% RSLogix 500 project Conveyor Belt with Order Fullfillment.RSS, saved by version 8.30.00.16 %
PROJECT "UNTITLED"    % processor: Bul.1763 MicroLogix 1100 Series B %

PROGRAM FILES
  LAD 2 "MAIN"  6 rungs
  LAD 3 "INPUTS"  7 rungs
  LAD 4 "OUTPUTS"  4 rungs
  LAD 5 "CONTROLS"  16 rungs

DATA FILES
  O0 OUTPUT  4 elements
  I1 INPUT  6 elements
  S2 STATUS  66 elements
  B3 BINARY  2 elements
  T4 TIMER  3 elements
  C5 COUNTER  1 elements
  R6 CONTROL  1 elements
  N7 INTEGER  3 elements
  F8 FLOAT  1 elements

LADDER 2 "MAIN"
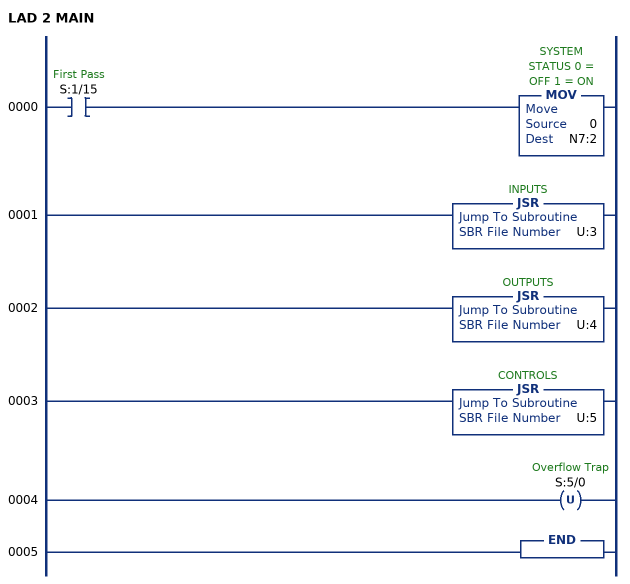
% Rung: 0 %
SOR XIC S:1/15 MOV 0 N7:2 EOR
%   S:1/15  "First Pass" %
%   N7:2  "SYSTEM STATUS 0 = OFF 1 = ON" %
% Rung: 1 %
SOR JSR U:3 EOR
%   U:3  "INPUTS" %
% Rung: 2 %
SOR JSR U:4 EOR
%   U:4  "OUTPUTS" %
% Rung: 3 %
SOR JSR U:5 EOR
%   U:5  "CONTROLS" %
% Rung: 4 %
SOR OTU S:5/0 EOR
%   S:5/0  "Overflow Trap" %
% Rung: 5 %
SOR END EOR

LADDER 3 "INPUTS"
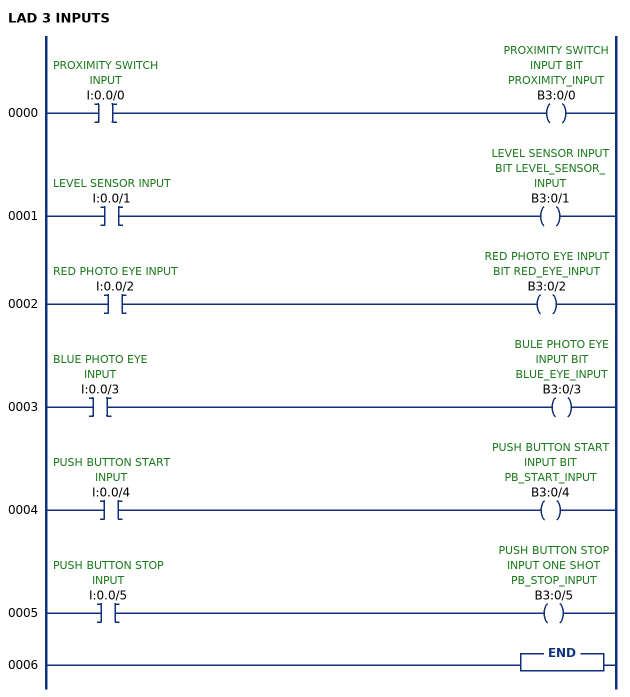
% Rung: 0 %
SOR XIC I:0.0/0 OTE B3:0/0 EOR
%   I:0.0/0  "PROXIMITY SWITCH INPUT" %
%   B3:0/0  PROXIMITY_INPUT  "PROXIMITY SWITCH INPUT BIT" %
% Rung: 1 %
SOR XIC I:0.0/1 OTE B3:0/1 EOR
%   I:0.0/1  "LEVEL SENSOR INPUT" %
%   B3:0/1  LEVEL_SENSOR_INPUT  "LEVEL SENSOR INPUT BIT" %
% Rung: 2 %
SOR XIC I:0.0/2 OTE B3:0/2 EOR
%   I:0.0/2  "RED PHOTO EYE INPUT" %
%   B3:0/2  RED_EYE_INPUT  "RED PHOTO EYE INPUT BIT" %
% Rung: 3 %
SOR XIC I:0.0/3 OTE B3:0/3 EOR
%   I:0.0/3  "BLUE PHOTO EYE INPUT" %
%   B3:0/3  BLUE_EYE_INPUT  "BULE PHOTO EYE INPUT BIT" %
% Rung: 4 %
SOR XIC I:0.0/4 OTE B3:0/4 EOR
%   I:0.0/4  "PUSH BUTTON START INPUT" %
%   B3:0/4  PB_START_INPUT  "PUSH BUTTON START INPUT BIT" %
% Rung: 5 %
SOR XIC I:0.0/5 OTE B3:0/5 EOR
%   I:0.0/5  "PUSH BUTTON STOP INPUT" %
%   B3:0/5  PB_STOP_INPUT  "PUSH BUTTON STOP INPUT ONE SHOT" %
% Rung: 6 %
SOR END EOR

LADDER 4 "OUTPUTS"
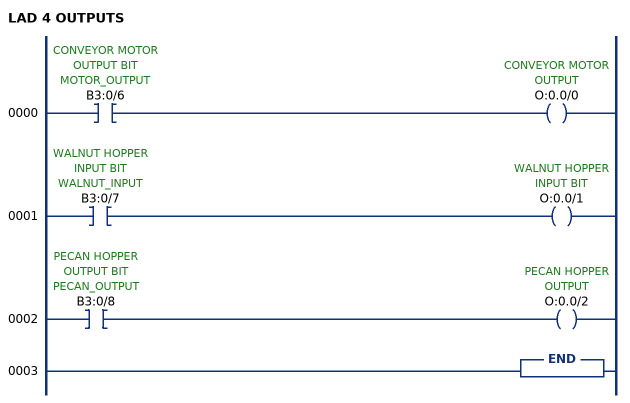
% Rung: 0 %
SOR XIC B3:0/6 OTE O:0.0/0 EOR
%   B3:0/6  MOTOR_OUTPUT  "CONVEYOR MOTOR OUTPUT BIT" %
%   O:0.0/0  "CONVEYOR MOTOR OUTPUT" %
% Rung: 1 %
SOR XIC B3:0/7 OTE O:0.0/1 EOR
%   B3:0/7  WALNUT_INPUT  "WALNUT HOPPER INPUT BIT" %
%   O:0.0/1  "WALNUT HOPPER INPUT BIT" %
% Rung: 2 %
SOR XIC B3:0/8 OTE O:0.0/2 EOR
%   B3:0/8  PECAN_OUTPUT  "PECAN HOPPER OUTPUT BIT" %
%   O:0.0/2  "PECAN HOPPER OUTPUT" %
% Rung: 3 %
SOR END EOR

LADDER 5 "CONTROLS"
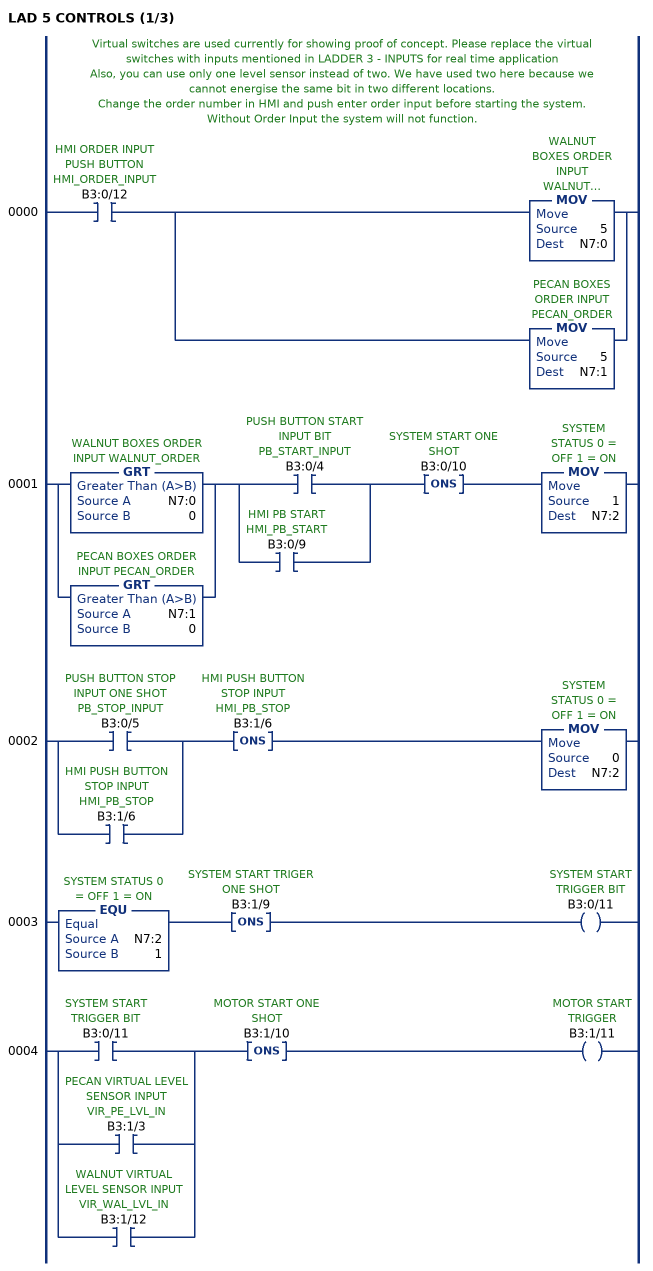
% Rung: 0 %
% Virtual switches are used currently for showing proof of concept. Please replace the virtual switches with inputs mentioned in LADDER 3 - INPUTS for real time application
% Also, you can use only one level sensor instead of two. We have used two here because we cannot energise the same bit in two different locations.
% 
% Change the order number in HMI and push enter order input before starting the system. Without Order Input the system will not function. %
SOR XIC B3:0/12 BST MOV 5 N7:0 NXB MOV 5 N7:1 BND EOR
%   B3:0/12  HMI_ORDER_INPUT  "HMI ORDER INPUT PUSH BUTTON" %
%   N7:0  WALNUT_ORDER  "WALNUT BOXES ORDER INPUT" %
%   N7:1  PECAN_ORDER  "PECAN BOXES ORDER INPUT" %
% Rung: 1 %
SOR BST GRT N7:0 0 NXB GRT N7:1 0 BND BST XIC B3:0/4 NXB XIC B3:0/9 BND ONS B3:0/10 MOV 1 N7:2 EOR
%   N7:0  WALNUT_ORDER  "WALNUT BOXES ORDER INPUT" %
%   N7:1  PECAN_ORDER  "PECAN BOXES ORDER INPUT" %
%   B3:0/4  PB_START_INPUT  "PUSH BUTTON START INPUT BIT" %
%   B3:0/9  HMI_PB_START  "HMI PB START" %
%   B3:0/10  "SYSTEM START ONE SHOT" %
%   N7:2  "SYSTEM STATUS 0 = OFF 1 = ON" %
% Rung: 2 %
SOR BST XIC B3:0/5 NXB XIC B3:1/6 BND ONS B3:1/6 MOV 0 N7:2 EOR
%   B3:0/5  PB_STOP_INPUT  "PUSH BUTTON STOP INPUT ONE SHOT" %
%   B3:1/6  HMI_PB_STOP  "HMI PUSH BUTTON STOP INPUT" %
%   N7:2  "SYSTEM STATUS 0 = OFF 1 = ON" %
% Rung: 3 %
SOR EQU N7:2 1 ONS B3:1/9 OTE B3:0/11 EOR
%   N7:2  "SYSTEM STATUS 0 = OFF 1 = ON" %
%   B3:1/9  "SYSTEM START TRIGER ONE SHOT" %
%   B3:0/11  "SYSTEM START TRIGGER BIT" %
% Rung: 4 %
SOR BST XIC B3:0/11 NXB XIC B3:1/3 NXB XIC B3:1/12 BND ONS B3:1/10 OTE B3:1/11 EOR
%   B3:0/11  "SYSTEM START TRIGGER BIT" %
%   B3:1/3  VIR_PE_LVL_IN  "PECAN VIRTUAL LEVEL SENSOR INPUT" %
%   B3:1/12  VIR_WAL_LVL_IN  "WALNUT VIRTUAL LEVEL SENSOR INPUT" %
%   B3:1/10  "MOTOR START ONE SHOT" %
%   B3:1/11  "MOTOR START TRIGGER" %

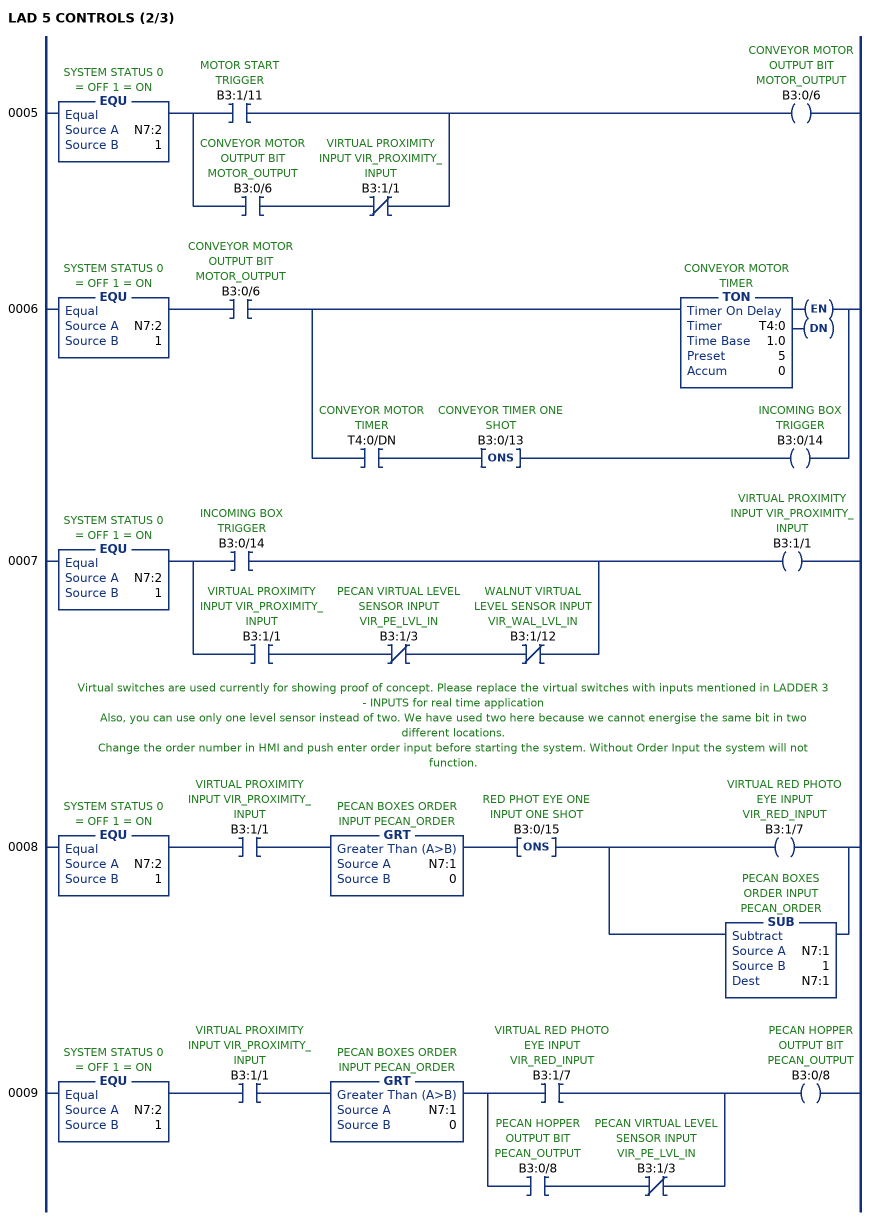
% Rung: 5 %
SOR EQU N7:2 1 BST XIC B3:1/11 NXB XIC B3:0/6 XIO B3:1/1 BND OTE B3:0/6 EOR
%   N7:2  "SYSTEM STATUS 0 = OFF 1 = ON" %
%   B3:1/11  "MOTOR START TRIGGER" %
%   B3:0/6  MOTOR_OUTPUT  "CONVEYOR MOTOR OUTPUT BIT" %
%   B3:1/1  VIR_PROXIMITY_INPUT  "VIRTUAL PROXIMITY INPUT" %
% Rung: 6 %
SOR EQU N7:2 1 XIC B3:0/6 BST TON T4:0 1.0 5 0 NXB XIC T4:0/DN ONS B3:0/13 OTE B3:0/14 BND EOR
%   N7:2  "SYSTEM STATUS 0 = OFF 1 = ON" %
%   B3:0/6  MOTOR_OUTPUT  "CONVEYOR MOTOR OUTPUT BIT" %
%   T4:0  "CONVEYOR MOTOR TIMER" %
%   B3:0/13  "CONVEYOR TIMER ONE SHOT" %
%   B3:0/14  "INCOMING BOX TRIGGER" %
% Rung: 7 %
SOR EQU N7:2 1 BST XIC B3:0/14 NXB XIC B3:1/1 XIO B3:1/3 XIO B3:1/12 BND OTE B3:1/1 EOR
%   N7:2  "SYSTEM STATUS 0 = OFF 1 = ON" %
%   B3:0/14  "INCOMING BOX TRIGGER" %
%   B3:1/1  VIR_PROXIMITY_INPUT  "VIRTUAL PROXIMITY INPUT" %
%   B3:1/3  VIR_PE_LVL_IN  "PECAN VIRTUAL LEVEL SENSOR INPUT" %
%   B3:1/12  VIR_WAL_LVL_IN  "WALNUT VIRTUAL LEVEL SENSOR INPUT" %
% Rung: 8 %
% Virtual switches are used currently for showing proof of concept. Please replace the virtual switches with inputs mentioned in LADDER 3 - INPUTS for real time application
% Also, you can use only one level sensor instead of two. We have used two here because we cannot energise the same bit in two different locations.
% 
% Change the order number in HMI and push enter order input before starting the system. Without Order Input the system will not function. %
SOR EQU N7:2 1 XIC B3:1/1 GRT N7:1 0 ONS B3:0/15 BST OTE B3:1/7 NXB SUB N7:1 1 N7:1 BND EOR
%   N7:2  "SYSTEM STATUS 0 = OFF 1 = ON" %
%   B3:1/1  VIR_PROXIMITY_INPUT  "VIRTUAL PROXIMITY INPUT" %
%   N7:1  PECAN_ORDER  "PECAN BOXES ORDER INPUT" %
%   B3:0/15  "RED PHOT EYE ONE INPUT ONE SHOT" %
%   B3:1/7  VIR_RED_INPUT  "VIRTUAL RED PHOTO EYE INPUT" %
% Rung: 9 %
SOR EQU N7:2 1 XIC B3:1/1 GRT N7:1 0 BST XIC B3:1/7 NXB XIC B3:0/8 XIO B3:1/3 BND OTE B3:0/8 EOR
%   N7:2  "SYSTEM STATUS 0 = OFF 1 = ON" %
%   B3:1/1  VIR_PROXIMITY_INPUT  "VIRTUAL PROXIMITY INPUT" %
%   N7:1  PECAN_ORDER  "PECAN BOXES ORDER INPUT" %
%   B3:1/7  VIR_RED_INPUT  "VIRTUAL RED PHOTO EYE INPUT" %
%   B3:0/8  PECAN_OUTPUT  "PECAN HOPPER OUTPUT BIT" %
%   B3:1/3  VIR_PE_LVL_IN  "PECAN VIRTUAL LEVEL SENSOR INPUT" %

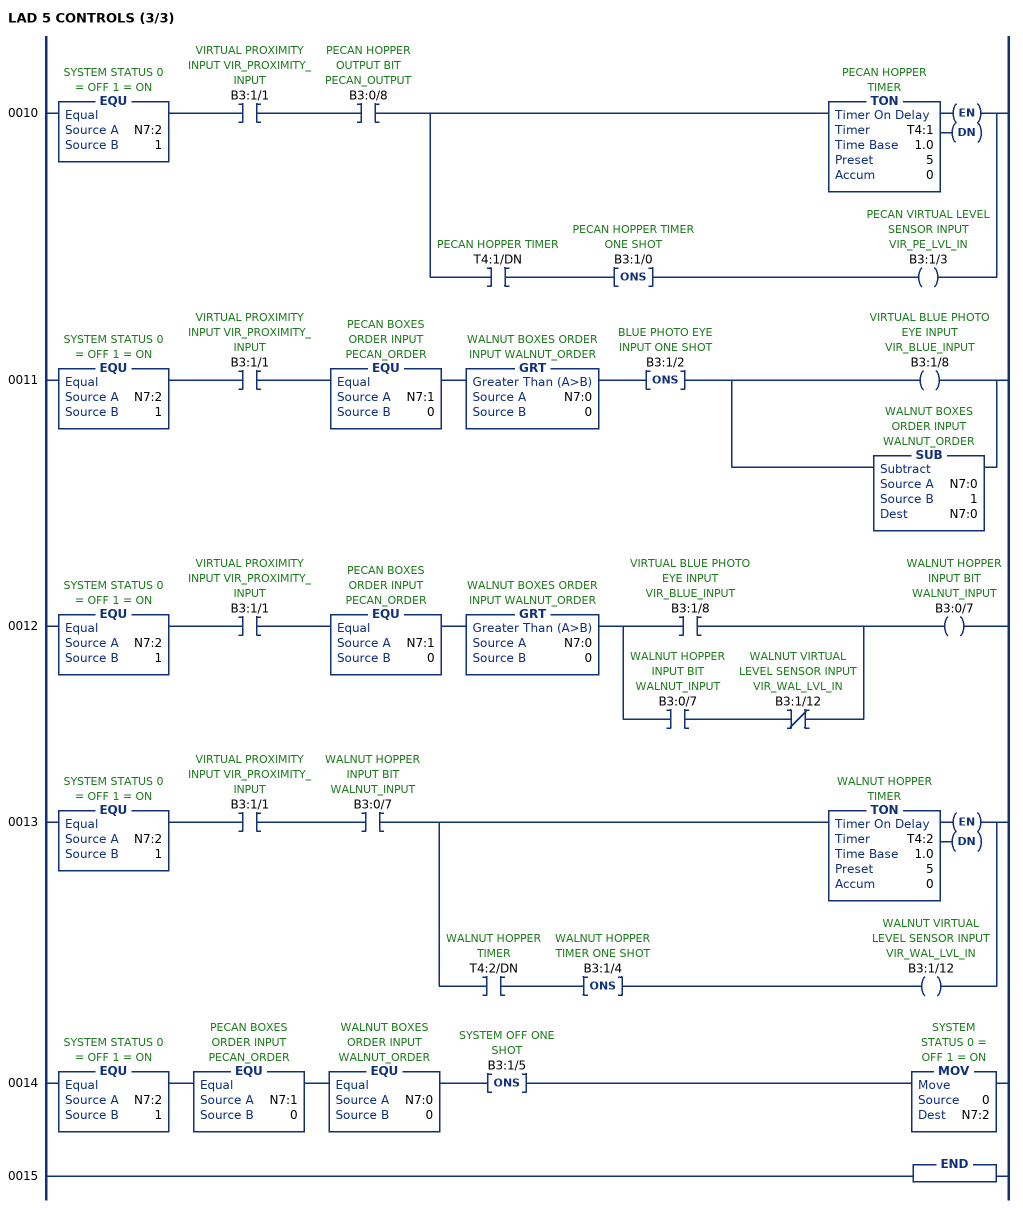
% Rung: 10 %
SOR EQU N7:2 1 XIC B3:1/1 XIC B3:0/8 BST TON T4:1 1.0 5 0 NXB XIC T4:1/DN ONS B3:1/0 OTE B3:1/3 BND EOR
%   N7:2  "SYSTEM STATUS 0 = OFF 1 = ON" %
%   B3:1/1  VIR_PROXIMITY_INPUT  "VIRTUAL PROXIMITY INPUT" %
%   B3:0/8  PECAN_OUTPUT  "PECAN HOPPER OUTPUT BIT" %
%   T4:1  "PECAN HOPPER TIMER" %
%   B3:1/0  "PECAN HOPPER TIMER ONE SHOT" %
%   B3:1/3  VIR_PE_LVL_IN  "PECAN VIRTUAL LEVEL SENSOR INPUT" %
% Rung: 11 %
SOR EQU N7:2 1 XIC B3:1/1 EQU N7:1 0 GRT N7:0 0 ONS B3:1/2 BST OTE B3:1/8 NXB SUB N7:0 1 N7:0 BND EOR
%   N7:2  "SYSTEM STATUS 0 = OFF 1 = ON" %
%   B3:1/1  VIR_PROXIMITY_INPUT  "VIRTUAL PROXIMITY INPUT" %
%   N7:1  PECAN_ORDER  "PECAN BOXES ORDER INPUT" %
%   N7:0  WALNUT_ORDER  "WALNUT BOXES ORDER INPUT" %
%   B3:1/2  "BLUE PHOTO EYE INPUT ONE SHOT" %
%   B3:1/8  VIR_BLUE_INPUT  "VIRTUAL BLUE PHOTO EYE INPUT" %
% Rung: 12 %
SOR EQU N7:2 1 XIC B3:1/1 EQU N7:1 0 GRT N7:0 0 BST XIC B3:1/8 NXB XIC B3:0/7 XIO B3:1/12 BND OTE B3:0/7 EOR
%   N7:2  "SYSTEM STATUS 0 = OFF 1 = ON" %
%   B3:1/1  VIR_PROXIMITY_INPUT  "VIRTUAL PROXIMITY INPUT" %
%   N7:1  PECAN_ORDER  "PECAN BOXES ORDER INPUT" %
%   N7:0  WALNUT_ORDER  "WALNUT BOXES ORDER INPUT" %
%   B3:1/8  VIR_BLUE_INPUT  "VIRTUAL BLUE PHOTO EYE INPUT" %
%   B3:0/7  WALNUT_INPUT  "WALNUT HOPPER INPUT BIT" %
%   B3:1/12  VIR_WAL_LVL_IN  "WALNUT VIRTUAL LEVEL SENSOR INPUT" %
% Rung: 13 %
SOR EQU N7:2 1 XIC B3:1/1 XIC B3:0/7 BST TON T4:2 1.0 5 0 NXB XIC T4:2/DN ONS B3:1/4 OTE B3:1/12 BND EOR
%   N7:2  "SYSTEM STATUS 0 = OFF 1 = ON" %
%   B3:1/1  VIR_PROXIMITY_INPUT  "VIRTUAL PROXIMITY INPUT" %
%   B3:0/7  WALNUT_INPUT  "WALNUT HOPPER INPUT BIT" %
%   T4:2  "WALNUT HOPPER TIMER" %
%   B3:1/4  "WALNUT HOPPER TIMER ONE SHOT" %
%   B3:1/12  VIR_WAL_LVL_IN  "WALNUT VIRTUAL LEVEL SENSOR INPUT" %
% Rung: 14 %
SOR EQU N7:2 1 EQU N7:1 0 EQU N7:0 0 ONS B3:1/5 MOV 0 N7:2 EOR
%   N7:2  "SYSTEM STATUS 0 = OFF 1 = ON" %
%   N7:1  PECAN_ORDER  "PECAN BOXES ORDER INPUT" %
%   N7:0  WALNUT_ORDER  "WALNUT BOXES ORDER INPUT" %
%   B3:1/5  "SYSTEM OFF ONE SHOT" %
% Rung: 15 %
SOR END EOR

OTHER DOCUMENTED ADDRESSES
  U:6  "ALARMS"

DATA TABLE (non-zero values as saved)
DATA T4
% .PRE .ACC %
% T4:0 % 5 0
% T4:1 % 5 0
% T4:2 % 5 0
